    //=================================================================
    // 16 - Stack buffer conveyors
    //=================================================================

    // EN: Common speed reference for all stack buffer conveyors [m/min].
    // PT: Referência comum de velocidade para todas as esteiras buffer [m/min].
    stackBufferConveyorsSpeedMPM               : REAL := 20.0;

    // EN: Additional running time after the target sensor is activated
    //     on buffer conveyors 1 and 2. Conveyor 3 stops immediately.
    // PT: Tempo adicional de movimento após o acionamento do sensor alvo
    //     nas esteiras buffer 1 e 2. A esteira 3 para imediatamente.
    stackBufferConveyorsStopDelay              : TIME := T#500MS;

    // EN: Maximum time allowed to transfer a stack to a buffer position.
    // PT: Tempo máximo permitido para transferir uma pilha até uma posição buffer.
    stackBufferTransferTimeout                 : TIME := T#30S;

    // EN: Time with all buffer positions occupied before requesting
    //     a machine speed reduction.
    // PT: Tempo com todas as posições buffer ocupadas antes de solicitar
    //     a redução da velocidade da máquina.
    stackBufferFullSpeedReductionDelay         : TIME := T#10S;

	//==============================================================
	// Configuration parameters / Parâmetros de configuração
	//==============================================================
	paperPressOnTime  : TIME := T#2S;
	paperPressOffTime : TIME := T#6S;

    //=================================================================
    // 17 - EN: Elevator servo controlled shutdown
    //      PT: Desligamento controlado do servo do elevador
    //=================================================================

    // EN: Time to keep the elevator servo enabled while quick stop is processed.
    // PT: Tempo para manter o servo do elevador habilitado durante o processamento do quick stop.
    elevatorDriveDisableDelay          : TIME := T#500MS;

    //=================================================================
    // 18 - Sheet conveyor 1 exhaust fan
    //=================================================================

    // EN: Minimum line speed required to run the exhaust fan [m/min].
    // PT: Velocidade mínima da linha necessária para ligar o exaustor [m/min].
    sheetConveyor1ExhaustFanLineSpeedThresholdMPM : REAL := 10.0;

    // EN: Time to keep the exhaust fan running after line speed drops
    //     to or below the configured threshold.
    // PT: Tempo para manter o exaustor ligado após a velocidade da linha cair
    //     até ou abaixo do limite configurado.
    sheetConveyor1ExhaustFanStopDelay              : TIME := T#10S;

END_STRUCT
END_TYPE

// ---- Library/Machine/Stacker/Cpx/DataTypes/hmiAlarmsComplexStacker_TypeStruct.TcDUT
TYPE hmiAlarmsComplexStacker_TypeStruct :
STRUCT

    //==============================================================
    // General / system alarms
    //==============================================================
    safetyCircuitNotOk                 : BOOL;
    systemFaultActive                  : BOOL;
    systemNotEnabled                   : BOOL;

    // EN: Generic safety feedback diagnostic alarms.
    // PT: Alarmes genéricos de diagnóstico dos retornos de segurança.
    safetyFeedback1NotOk               : BOOL;
    safetyFeedback2NotOk               : BOOL;
    safetyFeedback3NotOk               : BOOL;
    safetyFeedback4NotOk               : BOOL;
    safetyFeedback5NotOk               : BOOL;
    safetyFeedback6NotOk               : BOOL;
    safetyFeedback7NotOk               : BOOL;
    safetyFeedback8NotOk               : BOOL;

    //==============================================================
    // Sheet conveyor group alarms
    //==============================================================
    sheetConveyor1DriveNotOk           : BOOL;
    sheetConveyor2DriveNotOk           : BOOL;
    sheetConveyor3DriveNotOk           : BOOL;
    sheetConveyor4DriveNotOk           : BOOL;
    sheetConveyorGroupFault            : BOOL;
    synchronizedConveyorsNotRunning    : BOOL;

    //==============================================================
    // EN: Stack buffer conveyor alarms
    // PT: Alarmes das esteiras buffer de pilhas
    //==============================================================
    stackBufferConveyor1DriveNotOk      : BOOL;
    stackBufferConveyor2DriveNotOk      : BOOL;
    stackBufferConveyor3DriveNotOk      : BOOL;
    stackBufferConveyorGroupFault       : BOOL;

    // EN: Automatic stack transfer exceeded the configured timeout.
    // PT: A transferência automática da pilha excedeu o timeout configurado.
    stackBufferTransferTimeout          : BOOL;

    // EN: All three stack buffer positions are occupied.
    // PT: As três posições do buffer de pilhas estão ocupadas.
    stackBufferFull                     : BOOL;

    // EN: Machine speed reduction was requested because the buffer stayed full.
    // PT: A redução de velocidade da máquina foi solicitada porque o buffer permaneceu cheio.
    stackBufferSpeedReductionActive     : BOOL;

    //==============================================================
    // Sheet stack separation alarms / indications
    //==============================================================
    sheetStackSeparationNotReady       : BOOL;
    sheetStackSeparationActive         : BOOL;
    sheetStackBrakeActive              : BOOL;

    //==============================================================
    // Sheet stack discharge sequence alarms / indications
    //==============================================================
    sheetStackDischargeFault           : BOOL;
    sheetStackDischargeLastCycleNotOk  : BOOL;
    sheetStackDischargeTimeout         : BOOL;
    sheetStackDischargeManualSkip      : BOOL;

    // EN: Detailed discharge sequence timeout alarms.
    // PT: Alarmes detalhados de timeout da sequência de descarte.
    sheetStackDischargeWaitSeparationTimeout : BOOL;
    sheetStackDischargePositioningTimeout    : BOOL;
    sheetStackDischargeConveyorStartTimeout  : BOOL;
    sheetStackDischargePlatformClearTimeout  : BOOL;
    sheetStackDischargeReturnTimeout         : BOOL;

    //==============================================================
    // Sheet stack discharge conveyor alarms
    //==============================================================
    sheetStackDischargeConveyorDriveNotOk : BOOL;
    sheetStackDischargeConveyorFault      : BOOL;

    //==============================================================
    // Backstop alarms / indications
    //==============================================================
    backstopDriveNotOk                 : BOOL;
    backstopFault                      : BOOL;
    backstopNotHomed                   : BOOL;
    backstopNotInPosition              : BOOL;

    // EN: Detailed backstop homing alarms.
    // PT: Alarmes detalhados do homing do backstop.
    backstopHomingTimeout              : BOOL;
    backstopInvalidHomeDirection       : BOOL;

    backstopSafeMaxLimitActive         : BOOL;
    backstopSafeMinLimitActive         : BOOL;
    backstopMaxLimitActive             : BOOL;
    backstopMinLimitActive             : BOOL;

    backstopManualInterventionActive   : BOOL;

    //==============================================================
    // Elevator alarms / indications
    //==============================================================
    elevatorDriveNotOk          : BOOL;
    elevatorFault               : BOOL;
    elevatorNotHomed            : BOOL;
    elevatorNotInPosition       : BOOL;

    // EN: Elevator homing exceeded the configured timeout.
    // PT: O homing do elevador excedeu o timeout configurado.
    elevatorHomingTimeout       : BOOL;

    // EN: An upward movement request is blocked by the backstop material sensor.
    // PT: Um pedido de subida está bloqueado pelo sensor de material do backstop.
    elevatorUpBlockedByBackstopMaterialInterlock : BOOL;

    elevatorUpperSafetyLimitActive : BOOL;
    elevatorLowerSafetyLimitActive : BOOL;
    elevatorUpperLimitActive       : BOOL;
    elevatorLowerLimitActive       : BOOL;

END_STRUCT
END_TYPE

// ---- Library/Machine/Stacker/Cpx/DataTypes/hmiCommandsComplexStacker_TypeStruct.TcDUT
TYPE hmiCommandsComplexStacker_TypeStruct :
STRUCT

    //==============================================================
    // EN: System master commands
    // PT: Comandos gerais do sistema
    //==============================================================
    // EN: Momentary master start command.
    // PT: Comando momentâneo de partida geral.
    startCmd                                : BOOL;

    // EN: Momentary master stop command.
    // PT: Comando momentâneo de parada geral.
    stopCmd                                 : BOOL;

    // EN: Momentary fault reset command.
    // PT: Comando momentâneo de reset das falhas.
    resetCmd                                : BOOL;

	blockConveyorCmd					: BOOL;

    //==============================================================
    // EN: Sheet conveyor group commands
    // PT: Comandos do grupo de esteiras de chapas
    //==============================================================
    // EN: Momentary speed-up command for the sheet conveyors.
    // PT: Comando momentâneo para acelerar as esteiras de chapas.
    sheetConveyorsSpeedUpCmd                : BOOL;


    //==============================================================
    // EN: Package and sheet handling commands
    // PT: Comandos de pacote e manuseio das chapas
    //==============================================================
    // EN: Momentary request to complete and discharge the current package.
    // PT: Solicitação momentânea para concluir e descarregar o pacote atual.
    packageCompleteCmd                      : BOOL;

    // EN: Command to lower the no-crush rollers.
    // PT: Comando para baixar os rolos no-crush.
    noCrushRollersDownCmd                   : BOOL;


    //==============================================================
    // EN: Elevator commands
    // PT: Comandos do elevador
    //==============================================================
    // EN: Maintained elevator automatic-mode command.
    // PT: Comando mantido do modo automático do elevador.
    elevatorAutoCmd                         : BOOL;

    // EN: Momentary elevator homing command.
    // PT: Comando momentâneo de homing do elevador.
    elevatorHomeCmd                         : BOOL;

    // EN: Hold-to-run elevator jog-up command.
    // PT: Comando de jog mantido para subir o elevador.
    elevatorUpCmd                           : BOOL;

    // EN: Hold-to-run elevator jog-down command.
    // PT: Comando de jog mantido para descer o elevador.
    elevatorDownCmd                         : BOOL;


    //==============================================================
    // EN: Backstop commands
    // PT: Comandos do backstop
    //==============================================================
    // EN: Maintained backstop automatic-mode command.
    // PT: Comando mantido do modo automático do backstop.
    backstopAutoCmd                         : BOOL;

    // EN: Momentary backstop homing command.
    // PT: Comando momentâneo de homing do backstop.
    backstopHomeCmd                         : BOOL;

    // EN: Momentary command to execute programmed backstop positioning.
    // PT: Comando momentâneo para executar o posicionamento programado do backstop.
    backstopExecutePositioningCmd           : BOOL;

    // EN: Hold-to-run command to open the backstop.
    // PT: Comando mantido de jog para abrir o backstop.
    backstopOpenCmd                         : BOOL;

    // EN: Hold-to-run command to close the backstop.
    // PT: Comando mantido de jog para fechar o backstop.
    backstopCloseCmd                        : BOOL;


    //==============================================================
    // EN: Discharge and stack buffer conveyor commands
    // PT: Comandos das esteiras de descarga e buffer de pilhas
    //==============================================================
    // EN: Hold-to-run manual command for the stack discharge conveyor.
    // PT: Comando manual mantido da esteira de descarga da pilha.
    sheetStackDischargeConveyorManualRunCmd : BOOL;

    // EN: Hold-to-run manual command for all stack buffer conveyors.
    // PT: Comando manual mantido para todas as esteiras buffer de pilhas.
    stackBufferConveyorsRunCmd              : BOOL;


    //==============================================================
    // EN: Auxiliary pneumatic commands
    // PT: Comandos pneumáticos auxiliares
    //==============================================================
    // EN: Enables the cyclic paper press operation.
    // PT: Habilita a operação cíclica do prensa-papel.
    paperPressAutoManCmd                    : BOOL;

    // EN: Enables automatic operation of the exhaust fan installed
    //     on sheet conveyor 1.
    // PT: Habilita a operação automática do exaustor instalado
    //     na esteira de chapas 1.
    sheetConveyor1ExhaustFanCmd             : BOOL;

    // EN: Enables the four independent sheet brush commands.
    // PT: Habilita os comandos independentes das quatro escovas de chapas.
    sheetBrushAutoManCmd                    : BOOL;

    // EN: Individual sheet brush commands.
    // PT: Comandos individuais das escovas de chapas.
    sheetBrush1Cmd                          : BOOL;
    sheetBrush2Cmd                          : BOOL;
    sheetBrush3Cmd                          : BOOL;
    sheetBrush4Cmd                          : BOOL;

END_STRUCT
END_TYPE

// ---- Library/Machine/Stacker/Cpx/DataTypes/hmiStatusComplexStacker_TypeStruct.TcDUT
TYPE hmiStatusComplexStacker_TypeStruct :
STRUCT

    //==============================================================
    // System general status
    //==============================================================
    systemRunEnable                         : BOOL;        // EN: Master system run enable
    safetyCircuitOk                         : BOOL;        // EN: Safety circuit status
    faultActive                             : BOOL;        // EN: General fault active
    deviceState                             : STRING(30);  // EN: General device state text


    //==============================================================
    // Sheet conveyor group status
    //==============================================================
    synchronizedConveyorsRunning            : BOOL;        // EN: All synchronized conveyors running

    sheetConveyor1Run                       : BOOL;        // EN: Sheet conveyor 1 run output
    sheetConveyor2Run                       : BOOL;        // EN: Sheet conveyor 2 run output
    sheetConveyor3Run                       : BOOL;        // EN: Sheet conveyor 3 run output
    sheetConveyor4Run                       : BOOL;        // EN: Sheet conveyor 4 run output

    sheetConveyor1SpeedRefMPM               : REAL;        // EN: Sheet conveyor 1 speed reference [m/min]
    sheetConveyor2SpeedRefMPM               : REAL;        // EN: Sheet conveyor 2 speed reference [m/min]
    sheetConveyor3SpeedRefMPM               : REAL;        // EN: Sheet conveyor 3 speed reference [m/min]
    sheetConveyor4SpeedRefMPM               : REAL;        // EN: Sheet conveyor 4 speed reference [m/min]

    syncConveyorsState                      : INT;         // EN: Synchronized conveyor group state code


    //==============================================================
    // Sheet stack separation status
    //==============================================================
    sheetStackSeparationReady               : BOOL;        // EN: Stack separation ready
    sheetStackSeparationActive              : BOOL;        // EN: Stack separation active
    sheetStackBrakeActive                   : BOOL;        // EN: Stack brake active

    sheetStackSeparationDistanceM           : REAL;        // EN: Current separation distance [m]
    sheetStackSeparationTargetDistanceM     : REAL;        // EN: Target separation distance [m]


    //==============================================================
    // Sheet stack discharge sequence status
    //==============================================================
    sheetStackDischargeState                : STRING(30);  // EN: Discharge sequence state text
    sheetStackDischargeStateCode            : INT;         // EN: Discharge sequence state code

    sheetStackDischargePending              : BOOL;        // EN: Discharge cycle pending
    sheetStackDischargeActive               : BOOL;        // EN: Discharge cycle active
    sheetStackDischargeStarted              : BOOL;        // EN: Discharge cycle started pulse/status
    sheetStackDischargeFinished             : BOOL;        // EN: Discharge cycle finished pulse/status

    sheetStackDischargeFault                : BOOL;        // EN: Discharge sequence fault
    sheetStackDischargeFaultCode            : INT;         // EN: Current discharge fault code

    sheetStackDischargeLastCycleOk          : BOOL;        // EN: Last discharge cycle completed successfully
    sheetStackDischargeLastResultCode       : INT;         // EN: Last discharge result code
    sheetStackDischargeLastFaultStepCode    : INT;         // EN: Last discharge fault step code
    sheetStackDischargeLastFaultCode        : INT;         // EN: Last discharge fault code


    //==============================================================
    // Sheet stack discharge conveyor status
    //==============================================================
    sheetStackDischargeConveyorState        : STRING(30);  // EN: Discharge conveyor state text
    sheetStackDischargeConveyorRun          : BOOL;        // EN: Discharge conveyor run output
    sheetStackDischargeConveyorSpeedRefMPM  : REAL;        // EN: Discharge conveyor speed reference [m/min]

    sheetStackDischargeConveyorFault        : BOOL;        // EN: Discharge conveyor fault
    sheetStackDischargeConveyorFaultCode    : INT;         // EN: Discharge conveyor fault code


    //==============================================================
    // Backstop status
    //==============================================================
    backstopState                           : STRING(30);  // EN: Backstop state text
    backstopHomed                           : BOOL;        // EN: Backstop homing completed
    backstopHomeRunning                     : BOOL;        // EN: Backstop homing sequence running
    backstopInPosition                      : BOOL;        // EN: Backstop is inside target tolerance

    backstopPositionMm                      : REAL;        // EN: Actual backstop position [mm]
    backstopTargetPositionMm                : REAL;        // EN: Active backstop target position [mm]
    backstopPositionErrorMm                 : REAL;        // EN: Backstop position error [mm]

    backstopRunFw                           : BOOL;        // EN: Backstop forward/open run output
    backstopRunRev                          : BOOL;        // EN: Backstop reverse/close run output
    backstopSpeedRefMmps                    : REAL;        // EN: Backstop speed reference [mm/s]

    backstopPlateUpSolenoid                 : BOOL;        // EN: Backstop plate up solenoid
    backstopSetEncoderPosition              : BOOL;        // EN: Backstop set encoder pulse
    backstopSetEncoderPositionMm            : REAL;        // EN: Backstop set encoder position [mm]

    backstopManualInterventionActive        : BOOL;        // EN: Manual intervention memory active
    backstopManualInterventionPositionMm    : REAL;        // EN: Stored manual intervention position [mm]

    backstopFault                           : BOOL;        // EN: Backstop fault
    backstopFaultCode                       : INT;         // EN: Backstop fault code


    //==============================================================
    // Elevator status
    //==============================================================
    elevatorState                    : STRING(30);  // EN: Elevator state text
    elevatorHomed                    : BOOL;        // EN: Elevator homing completed
    elevatorInPosition               : BOOL;        // EN: Elevator is inside target tolerance

    elevatorPositionMm               : REAL;        // EN: Actual elevator position [mm]
    elevatorTargetPositionMm         : REAL;        // EN: Active elevator target position [mm]
    elevatorPositionErrorMm          : REAL;        // EN: Elevator position error [mm]

    elevatorRunUp                    : BOOL;        // EN: Elevator up run output
    elevatorRunDown                  : BOOL;        // EN: Elevator down run output
    elevatorBrakeRelease             : BOOL;        // EN: Elevator brake release output

    // EN: Elevator servo enable and quick-stop outputs.
    // PT: Saídas de habilitação e quick stop do servo do elevador.
    elevatorDriveEnable               : BOOL;
    elevatorQuickStop                 : BOOL;

    elevatorSpeedRefMmps             : REAL;        // EN: Elevator speed reference [mm/s]

    elevatorSetEncoderPosition       : BOOL;        // EN: Elevator set encoder pulse
    elevatorSetEncoderPositionMm     : REAL;        // EN: Elevator set encoder position [mm]

    elevatorFault                    : BOOL;        // EN: Elevator fault
    elevatorFaultCode                : INT;         // EN: Elevator fault code


    //==============================================================
    // EN: Auxiliary pneumatic output status
    // PT: Estados das saídas pneumáticas auxiliares
    //==============================================================
    // EN: Paper press solenoid output.
    // PT: Saída do solenoide do prensa-papel.
    paperPressSolenoid                      : BOOL;

    // EN: Sheet conveyor 1 exhaust fan run output.
    // PT: Saída de acionamento do exaustor da esteira de chapas 1.
    sheetConveyor1ExhaustFanRun             : BOOL;

    // EN: Sheet brush valve outputs.
    // PT: Saídas das válvulas das escovas de chapas.
    sheetBrush1Valve                        : BOOL;
    sheetBrush2Valve                        : BOOL;
    sheetBrush3Valve                        : BOOL;
    sheetBrush4Valve                        : BOOL;


    //==============================================================
    // Process values
    //==============================================================
    lineSpeedMPM                            : REAL;        // EN: Current line speed [m/min]
    sheetLengthMm                           : REAL;        // EN: Current sheet length [mm]
    stackHeightMm                           : REAL;        // EN: Current stack height [mm]


    //==============================================================
    // Input / drive status mirror
    //==============================================================
    sheetConveyor1DriveOk                   : BOOL;        // EN: Sheet conveyor 1 drive OK
    sheetConveyor2DriveOk                   : BOOL;        // EN: Sheet conveyor 2 drive OK
    sheetConveyor3DriveOk                   : BOOL;        // EN: Sheet conveyor 3 drive OK
    sheetConveyor4DriveOk                   : BOOL;        // EN: Sheet conveyor 4 drive OK

    backstopDriveOk                         : BOOL;        // EN: Backstop drive OK
    elevatorDriveOk                  : BOOL;        // EN: Elevator drive OK
    sheetStackDischargeConveyorDriveOk      : BOOL;        // EN: Discharge conveyor drive OK

END_STRUCT
END_TYPE

// ---- Library/Machine/Stacker/Simple/DataTypes/SimpleStackerConfig_TypeStruct.TcDUT
TYPE SimpleStackerConfig_TypeStruct :
STRUCT

    //=================================================================
    // 01 - General line / stacker speed configuration
    //=================================================================

    // EN: Normal stacker speed ratio relative to line speed.
    //     Example: 0.17 = stacker runs at 17% of line speed.
    // PT: Fator normal de velocidade do stacker em relação à velocidade da linha.
    //     Exemplo: 0.17 = stacker trabalha com 17% da velocidade da linha.
    stackerSpeedRatio                         : REAL := 0.17;

    // EN: Minimum and maximum speed reference allowed for sheet conveyors [m/min].
    // PT: Referência mínima e máxima permitida para as esteiras de chapas [m/min].
    minimumSpeedMPM                           : REAL := 10.0;
    maximumSpeedMPM                           : REAL := 80.0;

    // EN: Maximum ramp velocity for conveyor speed references [m/min/s].
    // PT: Velocidade máxima da rampa para referências das esteiras [m/min/s].
    rampVelocityUpMaxMPMps                    : REAL := 1000.0;
    rampVelocityDownMaxMPMps                  : REAL := 1000.0;

    // EN: Ramp acceleration / deceleration used by S-ramp smoothing [m/min/s²].
    // PT: Aceleração / desaceleração usada na suavização da rampa S [m/min/s²].
    rampAccelerationUpMPMps2                  : REAL := 1000.0;
    rampAccelerationDownMPMps2                : REAL := 1000.0;


    //=================================================================
    // 02 - Sheet conveyor group: speed trim and mechanical length
    //=================================================================

    // EN: Individual speed trim for each synchronized sheet conveyor.
    //     1.0 = no correction.
    // PT: Correção individual de velocidade para cada esteira sincronizada.
    //     1.0 = sem correção.
    sheetConveyor1SpeedTrim                   : REAL := 1.0;
    sheetConveyor2SpeedTrim                   : REAL := 1.0;
    sheetConveyor3SpeedTrim                   : REAL := 1.0;

    // EN: Sheet conveyor mechanical length [m].
    // PT: Comprimento mecânico da esteira de chapas [m].
    sheetConveyor1LengthM                     : REAL := 1.85;
    sheetConveyor2LengthM                     : REAL := 1.0;
    sheetConveyor3LengthM                     : REAL := 2.0;

    // EN: Additional speed reference applied to sheet conveyors 1, 2 and 3
    //     when the external speed-up command is active [m/min].
    // PT: Referência adicional aplicada nas esteiras 1, 2 e 3
    //     quando o comando externo de aceleração estiver ativo [m/min].
    sheetConveyorsSpeedUpMPM                  : REAL := 20.0;


    //=================================================================
    // 03 - Sheet conveyor group: package separation
    //=================================================================

    // EN: Speed multiplier used during package separation.
    //     Example: 1.50 = 50% faster than normal speed.
    // PT: Multiplicador de velocidade usado durante a separação de pacote.
    //     Exemplo: 1.50 = 50% acima da velocidade normal.
    packageGapSpeedRatio                      : REAL := 3.0;

    // EN: Additional fixed speed offset during package separation [m/min].
    // PT: Offset fixo adicional de velocidade durante a separação de pacote [m/min].
    packageGapSpeedOffsetMPM                  : REAL := 0.0;

    // EN: Minimum line speed used as the conveyor speed calculation reference
    //     while package separation is active [m/min].
    //     Set to 0.0 to keep the actual line speed without a discharge override.
    // PT: Velocidade mínima da linha usada como referência para o cálculo das
    //     esteiras enquanto a separação da pilha estiver ativa [m/min].
    //     Usar 0.0 para manter a velocidade real da linha sem sobreposição no descarte.
    packageDischargeLineSpeedThresholdMPM     : REAL := 0.0;

    // EN: Minimum valid differential speed used for separation tracking [m/min].
    // PT: Velocidade diferencial mínima válida usada no rastreamento da separação [m/min].
    minimumOpeningSpeedMPM                    : REAL := 1.0;


    //=================================================================
    // 04 - Conveyor leveler: speed trim and position limits
    //=================================================================

    // EN: Individual speed trim for conveyor leveler synchronized movement.
    //     1.0 = no correction.
    // PT: Correção individual de velocidade para movimento sincronizado do nivelador.
    //     1.0 = sem correção.
    conveyorLevelerSpeedTrim                  : REAL := 1.0;

    // EN: Minimum and maximum allowed conveyor leveler position [mm].
    // PT: Posição mínima e máxima permitida para o nivelador da esteira [mm].
    conveyorLevelerMinPositionMm              : REAL := 10.0;
    conveyorLevelerMaxPositionMm              : REAL := 150.0;


    //=================================================================
    // 05 - Conveyor leveler: automatic positioning
    //=================================================================

    // EN: Offset added to stack height to calculate conveyor leveler target [mm].
    // PT: Offset somado à altura da pilha para calcular o alvo do nivelador [mm].
    conveyorLevelerStackHeightOffsetMm        : REAL := 0.0;

    // EN: Position tolerance to consider conveyor leveler in position [mm].
    // PT: Tolerância de posição para considerar o nivelador em posição [mm].
    conveyorLevelerPositionToleranceMm        : REAL := 2.0;

    // EN: Proportional gain for conveyor leveler position control [(mm/s)/mm].
    // PT: Ganho proporcional do controle de posição do nivelador [(mm/s)/mm].
    conveyorLevelerPositionKp                 : REAL := 5.0;

    // EN: Maximum speed allowed in automatic conveyor leveler positioning [mm/s].
    // PT: Velocidade máxima permitida no posicionamento automático do nivelador [mm/s].
    conveyorLevelerAutoMaxSpeedMmps           : REAL := 30.0;

    // EN: Minimum movement speed when the position error is above tolerance [mm/s].
    // PT: Velocidade mínima de movimento quando o erro de posição estiver acima da tolerância [mm/s].
    conveyorLevelerMinMoveSpeedMmps           : REAL := 5.0;


    //=================================================================
    // 06 - Conveyor leveler: manual movement
    //=================================================================

    // EN: Manual up/down speed for conveyor leveler [mm/s].
    // PT: Velocidade manual para subir/descer o nivelador da esteira [mm/s].
    conveyorLevelerManualSpeedMmps            : REAL := 50.0;

    // EN: Minimum speed reference required to enable conveyor leveler drive run [mm/s].
    // PT: Referência mínima de velocidade necessária para liberar RUN do acionamento do nivelador [mm/s].
    conveyorLevelerRunMinSpeedMmps            : REAL := 0.1;


    //=================================================================
    // 07 - Conveyor leveler: homing and encoder set
    //=================================================================

    // EN: Conveyor leveler homing speed [mm/s].
    // PT: Velocidade de homing do nivelador da esteira [mm/s].
    conveyorLevelerHomingSpeedMmps            : REAL := 30.0;

    // EN: Maximum allowed time for conveyor leveler homing movement.
    // PT: Tempo máximo permitido para o movimento de homing do nivelador.
    conveyorLevelerHomingTimeout              : TIME := T#30S;

    // EN: Pulse time for conveyor leveler encoder position set command.
    // PT: Tempo do pulso para comando de set da posição do encoder do nivelador.
    conveyorLevelerSetEncoderPulseTime        : TIME := T#200MS;


    //=================================================================
    // 08 - Conveyor leveler: magnetic brake
    //=================================================================

    // EN: Delay between brake release command and motor movement permission.
    // PT: Atraso entre o comando de liberação do freio e a permissão de movimento do motor.
    conveyorLevelerBrakeReleaseDelay          : TIME := T#300MS;

    // EN: Time to keep the brake released after movement stops.
    // PT: Tempo para manter o freio liberado após a parada do movimento.
    conveyorLevelerBrakeHoldTime              : TIME := T#2S;


    //=================================================================
    // 09 - Backstop: position limits
    //=================================================================

    // EN: Minimum and maximum allowed backstop position [mm].
    // PT: Posição mínima e máxima permitida para o backstop [mm].
    backstopMinPositionMm                     : REAL := 300.0;
    backstopMaxPositionMm                     : REAL := 5000.0;


    //=================================================================
    // 10 - Backstop: homing and encoder set
    //=================================================================

    // EN: Homing direction. -1 = close/min limit, +1 = open/max limit.
    // PT: Direção de homing. -1 = fechar/limite mínimo, +1 = abrir/limite máximo.
    backstopHomeDirection                     : INT := 1;

    // EN: Encoder position value to set after homing is completed [mm].
    // PT: Valor de posição gravado no encoder após finalizar o homing [mm].
    backstopHomePositionMm                    : REAL := 2985.0;

    // EN: Backstop homing speed [mm/s].
    // PT: Velocidade de homing do backstop [mm/s].
    backstopHomingSpeedMmps                   : REAL := 150.0;

    // EN: Maximum allowed time for backstop homing movement.
    // PT: Tempo máximo permitido para o movimento de homing do backstop.
    backstopHomingTimeout                     : TIME := T#40S;

    // EN: Pulse time for backstop encoder position set command.
    // PT: Tempo do pulso para comando de set da posição do encoder do backstop.
    backstopSetEncoderPulseTime               : TIME := T#200MS;


    //=================================================================
    // 11 - Backstop: automatic positioning
    //=================================================================

    // EN: Offset added to sheet length to calculate automatic backstop target [mm].
    // PT: Offset somado ao comprimento da chapa para calcular o alvo automático do backstop [mm].
    backstopSheetLengthOffsetMm               : REAL := 0.0;

    // EN: Position tolerance to consider the backstop in position [mm].
    // PT: Tolerância de posição para considerar o backstop em posição [mm].
    backstopPositionToleranceMm               : REAL := 5.0;

    // EN: Proportional gain for backstop position control [(mm/s)/mm].
    // PT: Ganho proporcional do controle de posição do backstop [(mm/s)/mm].
    backstopPositionKp                        : REAL := 3.0;

    // EN: Maximum speed allowed in automatic backstop positioning [mm/s].
    // PT: Velocidade máxima permitida no posicionamento automático do backstop [mm/s].
    backstopAutoMaxSpeedMmps                  : REAL := 400.0;

    // EN: Minimum movement speed when the position error is above tolerance [mm/s].
    // PT: Velocidade mínima de movimento quando o erro de posição estiver acima da tolerância [mm/s].
    backstopMinMoveSpeedMmps                  : REAL := 15.0;


    //=================================================================
    // 12 - Backstop: manual movement
    //=================================================================

    // EN: Manual open/close speed for backstop [mm/s].
    // PT: Velocidade manual para abrir/fechar o backstop [mm/s].
    backstopManualSpeedMmps                   : REAL := 80.0;

    // EN: Minimum speed reference required to enable backstop drive run [mm/s].
    // PT: Referência mínima de velocidade necessária para liberar RUN do acionamento do backstop [mm/s].
    backstopRunMinSpeedMmps                   : REAL := 10.0;


    //=================================================================
    // 13 - Sheet stack discharge conveyor
    //=================================================================

    // EN: Sheet stack discharge conveyor speed reference [m/min].
    // PT: Referência de velocidade da esteira de descarga da pilha [m/min].
    sheetStackDischargeConveyorSpeedMPM       : REAL := 70.0;

    // EN: Running time for sheet stack discharge conveyor.
    // PT: Tempo de giro da esteira de descarga da pilha.
    sheetStackDischargeTime                   : TIME := T#2S;


    //=================================================================
    // 14 - Sheet stack discharge sequence: backstop movement
    //=================================================================

    // EN: Additional backstop opening during sheet stack discharge [mm].
    // PT: Abertura adicional do backstop durante a descarga da pilha [mm].
    backstopDischargeOpenOffsetMm             : REAL := 100.0;


    //=================================================================
    // 15 - Sheet stack discharge sequence: step timeouts
    //=================================================================

    // EN: Maximum time to wait for package separation before discharge sequence continues.
    // PT: Tempo máximo de espera pela separação do pacote antes da sequência de descarga continuar.
    sheetStackDischargeWaitSeparationTimeout  : TIME := T#10S;

    // EN: Maximum time allowed for discharge positioning movement.
    // PT: Tempo máximo permitido para o movimento de posicionamento da descarga.
    sheetStackDischargePositioningTimeout     : TIME := T#10S;

    // EN: Maximum time allowed to confirm/start discharge conveyor movement.
    // PT: Tempo máximo permitido para confirmar/iniciar o movimento da esteira de descarga.
    sheetStackDischargeConveyorStartTimeout   : TIME := T#3S;

    // EN: Maximum time allowed for backstop return movement after discharge.
    // PT: Tempo máximo permitido para o retorno do backstop após a descarga.
    sheetStackDischargeReturnTimeout          : TIME := T#10S;

END_STRUCT
END_TYPE

// ---- Library/Machine/Stacker/Simple/DataTypes/SimpleStackerConfig_TypeStruct_1.TcDUT
TYPE SimpleStackerConfig_TypeStruct_1 :
STRUCT

    //==============================================================
    // Normal speed synchronization
    //==============================================================
    // EN: Normal stacker speed ratio relative to line speed.
    //     Example: 0.17 = stacker runs at 17% of line speed.
    // PT: Fator normal de velocidade do stacker em relação à linha.
    //     Exemplo: 0.17 = stacker trabalha com 17% da velocidade da linha.
    stackerSpeedRatio                 : REAL := 0.17;


    //==============================================================
    // Individual conveyor speed trim
    //==============================================================
    // EN: Individual speed correction for each conveyor.
    // PT: Correção individual de velocidade de cada esteira.
    sheetConveyor1SpeedTrim           : REAL := 1.0;
    sheetConveyor2SpeedTrim           : REAL := 1.0;
    sheetConveyor3SpeedTrim           : REAL := 1.0;
    conveyorLevelerSpeedTrim          : REAL := 1.0;

	//==============================================================
	// Sheet conveyors speed-up command
	//==============================================================
	// EN: Additional speed reference applied to sheet conveyors 1/2/3 [m/min].
	// PT: Referência adicional aplicada nas esteiras 1/2/3 [m/min].
	sheetConveyorsSpeedUpMPM : REAL := 20.0;
	
    //==============================================================
    // Conveyor length
    //==============================================================
    // EN: Conveyor length [m].
    // PT: Comprimento da esteira [m].
    sheetConveyor1LengthM             : REAL := 20.0;
    sheetConveyor2LengthM             : REAL := 20.0;
    sheetConveyor3LengthM             : REAL := 20.0;


    //==============================================================
    // Package separation
    //==============================================================
    // EN: Speed multiplier used during package separation.
    // PT: Multiplicador de velocidade usado durante a separação.
    packageGapSpeedRatio              : REAL := 1.50;

    // EN: Additional fixed speed offset during separation [m/min].
    // PT: Offset fixo adicional de velocidade durante a separação [m/min].
    packageGapSpeedOffsetMPM          : REAL := 0.0;

    // EN: Gap distance as factor of sheet length.
    //     Example: 0.25 with 2.0 m sheet = 0.5 m gap.
    // PT: Distância de abertura como fator do comprimento da chapa.
    //     Exemplo: 0.25 com chapa de 2.0 m = 0.5 m de vão.
//    packageGapLengthFactor            : REAL := 0.25;

    // EN: Minimum valid differential speed for opening calculation [m/min].
    // PT: Velocidade diferencial mínima válida para cálculo de abertura [m/min].
    minimumOpeningSpeedMPM            : REAL := 1.0;

    // EN: Maximum package gap distance allowed [m].
    // PT: Distância máxima permitida para abertura do pacote [m].
//    maximumPackageGapDistanceM        : REAL := 3.0;


    //==============================================================
    // Speed limits
    //==============================================================
    // EN: Minimum and maximum conveyor speed reference [m/min].
    // PT: Velocidade mínima e máxima de referência das esteiras [m/min].
    minimumSpeedMPM                   : REAL := 0.0;
    maximumSpeedMPM                   : REAL := 80.0;


    //==============================================================
    // Ramp parameters
    //==============================================================
    // EN: Maximum ramp velocity [m/min/s].
    // PT: Velocidade máxima da rampa [m/min/s].
    rampVelocityUpMaxMPMps            : REAL := 1000.0;
    rampVelocityDownMaxMPMps          : REAL := 1000.0;

    // EN: Ramp acceleration / S-ramp smoothing [m/min/s²].
    // PT: Aceleração da rampa / suavização da rampa S [m/min/s²].
    rampAccelerationUpMPMps2          : REAL := 1000.0;
    rampAccelerationDownMPMps2        : REAL := 1000.0;



	//==============================================================
	// Backstop homing
	//==============================================================
	// EN: Homing direction. -1 = close/min limit, +1 = open/max limit.
	// PT: Direção de homing. -1 = fechar/limite mínimo, +1 = abrir/limite máximo.
	backstopHomeDirection              : INT := -1;
	
	// EN: Encoder position value to set after homing is completed [mm].
	// PT: Valor de posição que será gravado no encoder após finalizar o homing [mm].
	backstopHomePositionMm             : REAL := 300.0;
	
	// EN: Backstop homing speed [mm/s].
	// PT: Velocidade de homing do backstop [mm/s].
	backstopHomingSpeedMmps            : REAL := 50.0;
	
	// EN: Maximum allowed time for homing movement.
	// PT: Tempo máximo permitido para o movimento de homing.
	backstopHomingTimeout              : TIME := T#30S;
	
	// EN: Pulse time for encoder position set command.
	// PT: Tempo do pulso para comando de set da posição do encoder.
	backstopSetEncoderPulseTime        : TIME := T#200MS;	
	//==============================================================
	// Backstop position limits
	//==============================================================
	// EN: Minimum allowed backstop position [mm].
	// PT: Posição mínima permitida do backstop [mm].
	backstopMinPositionMm              : REAL := 300.0;
	
	// EN: Maximum allowed backstop position [mm].
	// PT: Posição máxima permitida do backstop [mm].
	backstopMaxPositionMm              : REAL := 2500.0;
	
	
	//==============================================================
	// Backstop automatic positioning
	//==============================================================
	// EN: Offset added to sheet length to calculate automatic backstop target [mm].
	// PT: Offset somado ao comprimento da chapa para calcular o alvo automático [mm].
	backstopSheetLengthOffsetMm        : REAL := 0.0;
	
	// EN: Position tolerance to consider the backstop in position [mm].
	// PT: Tolerância de posição para considerar o backstop em posição [mm].
	backstopPositionToleranceMm        : REAL := 2.0;
	
	// EN: Proportional gain for position control [(mm/s)/mm].
	// PT: Ganho proporcional do controle de posição [(mm/s)/mm].
	backstopPositionKp                 : REAL := 0.5;
	
	// EN: Maximum speed allowed in automatic positioning [mm/s].
	// PT: Velocidade máxima permitida no posicionamento automático [mm/s].
	backstopAutoMaxSpeedMmps           : REAL := 150.0;
	
	// EN: Minimum movement speed when position error is above tolerance [mm/s].
	// PT: Velocidade mínima de movimento quando o erro de posição estiver acima da tolerância [mm/s].
	backstopMinMoveSpeedMmps           : REAL := 10.0;
	
	
	//==============================================================
	// Backstop manual movement
	//==============================================================
	// EN: Manual open/close speed [mm/s].
	// PT: Velocidade manual para abrir/fechar o backstop [mm/s].
	backstopManualSpeedMmps            : REAL := 80.0;
	
	// EN: Minimum speed reference to enable backstop drive run [mm/s].
	// PT: Referência mínima de velocidade para liberar RUN do inversor do backstop [mm/s].
	backstopRunMinSpeedMmps             : REAL := 0.1;
	
		
	//==============================================================
	// Conveyor leveler position limits
	//==============================================================
	conveyorLevelerMinPositionMm          : REAL := 0.0;
	conveyorLevelerMaxPositionMm          : REAL := 1000.0;
	
	
	//==============================================================
	// Conveyor leveler automatic control
	//==============================================================
	conveyorLevelerStackHeightOffsetMm    : REAL := 0.0;
	conveyorLevelerPositionToleranceMm    : REAL := 5.0;
	conveyorLevelerPositionKp             : REAL := 0.5;
	conveyorLevelerAutoMaxSpeedMmps       : REAL := 100.0;
	conveyorLevelerMinMoveSpeedMmps       : REAL := 5.0;
	
	
	//==============================================================
	// Conveyor leveler manual control
	//==============================================================
	conveyorLevelerManualSpeedMmps        : REAL := 50.0;
	
	
	//==============================================================
	// Conveyor leveler homing
	//==============================================================
	conveyorLevelerHomingSpeedMmps        : REAL := 30.0;
	conveyorLevelerHomingTimeout          : TIME := T#30S;
	
	
	//==============================================================
	// Conveyor leveler encoder set pulse
	//==============================================================
	conveyorLevelerSetEncoderPulseTime    : TIME := T#200MS;
	
	
	//==============================================================
	// Conveyor leveler magnetic brake
	//==============================================================
	conveyorLevelerBrakeReleaseDelay      : TIME := T#300MS;
	conveyorLevelerBrakeHoldTime          : TIME := T#2S;
	
	
	//==============================================================
	// Conveyor leveler drive enable
	//==============================================================
	conveyorLevelerRunMinSpeedMmps        : REAL := 0.1;	
	
	//==============================================================
	// Sheet stack discharge conveyor
	//==============================================================
	// EN: Discharge conveyor speed reference [m/min].
	// PT: Referência de velocidade da esteira de descarga [m/min].
	sheetStackDischargeConveyorSpeedMPM     : REAL := 20.0;
	
	// EN: Discharge conveyor running time.
	// PT: Tempo de giro da esteira de descarga.
	sheetStackDischargeTime                 : TIME := T#5S;
	
	
	//==============================================================
	// Backstop discharge movement
	//==============================================================
	// EN: Additional backstop opening during sheet stack discharge [mm].
	// PT: Abertura adicional do backstop durante a descarga da pilha [mm].
	backstopDischargeOpenOffsetMm           : REAL := 100.0;
	
	sheetStackDischargeWaitSeparationTimeout : TIME := T#10S;
	sheetStackDischargePositioningTimeout    : TIME := T#10S;
	sheetStackDischargeConveyorStartTimeout  : TIME := T#3S;
	sheetStackDischargeReturnTimeout         : TIME := T#10S;	
	
END_STRUCT
END_TYPE

// ---- Library/Machine/Stacker/Simple/E_BackstopState.TcDUT
{attribute 'qualified_only' := ''}
{attribute 'strict' := ''}
TYPE E_BackstopState :
(
	STOP := 0,
	HOME_FAST_SEARCH := 10,
	HOME_SLOW_EXIT_SENSOR := 11,
	HOME_SET_ENCODER := 12,
	HOME_WAIT_AFTER_SET := 13,
	HOME_MOVE_TO_TARGET := 14,
	MANUAL := 20,
	AUTO_POSITION := 30,
	FAULT := 40
);
END_TYPE

// ---- Library/Machine/Stacker/Simple/E_ConveyorLevelerState.TcDUT
{attribute 'qualified_only' := ''}
{attribute 'strict' := ''}
TYPE E_ConveyorLevelerState :
(
	STOP := 0,
	HOME_FAST_SEARCH := 10,
	HOME_SLOW_EXIT_SENSOR := 11,
	HOME_SET_ENCODER := 12,
	MANUAL := 20,
	AUTO_LEVELING := 30,
	FAULT := 40
);
END_TYPE

// ---- Library/Machine/Stacker/Simple/E_PackageSeparationState.TcDUT
{attribute 'qualified_only' := ''}
{attribute 'strict' := ''}
TYPE E_PackageSeparationState :
(
	NORMAL := 0,
	START_SEPARATION := 10,
	CONVEYOR_2_TRACKING := 20,
	CONVEYOR_3_TRACKING := 30,
	FINISH_SEPARATION := 40
);
END_TYPE

// ---- Library/Machine/Stacker/Simple/E_SheetStackDischargeState.TcDUT
{attribute 'qualified_only' := ''}
{attribute 'strict' := ''}
TYPE E_SheetStackDischargeState :
(
	IDLE := 0,
	WAIT_SEPARATION := 5,
	START_POSITIONING := 10,
	WAIT_BACKSTOP_POSITION := 20,
	DISCHARGING := 30,
	START_RETURN := 40,
	WAIT_BACKSTOP_RETURN := 50,
	FINISH := 60
);
END_TYPE

// ---- Library/Machine/Stacker/Simple/E_SyncConveyorsState.TcDUT
{attribute 'qualified_only' := ''}
{attribute 'strict' := ''}
TYPE E_SyncConveyorsState :
(
	IDLE := 0,
	RUN := 1,
	FAULT := 10
);
END_TYPE

// ---- Library/Sick/DT35-B15251 - Laser Sensor/DataTypes/_DT35B15251_DEV_CONFIG.TcDUT
TYPE _DT35B15251_DEV_CONFIG :
STRUCT

    //=============================================================
    // IO-Link process data
    //=============================================================

    processDataResolutionFactor : REAL := 1.0; 
    // 1.0 = process data in 1 mm steps
    // 0.1 = process data in 0.1 mm steps
    // 10.0 = process data in 10 mm steps


    //=============================================================
    // Distance limits
    //=============================================================

    distanceLowLimit  : REAL := 0.0;
    distanceHighLimit : REAL := 12000.0;


    //=============================================================
    // Relative distance from zero
    // EN: Shows distance starting from a configured zero point.
    // Example:
    // distance = 1500 mm
    // distanceZeroReference = 1000 mm
    // distanceFromZero = 500 mm
    //=============================================================

    distanceZeroReference       : REAL := 0.0;
    distanceFromZeroLowLimit    : REAL := 0.0;
    distanceFromZeroHighLimit   : REAL := 12000.0;


    //=============================================================
    // Height calculation
    // EN: Height is calculated from the measured distance.
    // Example:
    // heightReferenceDistance = distance from sensor to zero-height surface
    // height = heightReferenceDistance - distance
    //=============================================================

    heightReferenceDistance : REAL := 2000.0;
    heightLowLimit          : REAL := 0.0;
    heightHighLimit         : REAL := 2000.0;

END_STRUCT
END_TYPE

// ---- Library/Sick/DT35-B15251 - Laser Sensor/DataTypes/_DT35B15251_HWTOPLC_PDOS.TcDUT
TYPE _DT35B15251_HWTOPLC_PDOS :
STRUCT
	
	inputByte_0 	 : BYTE;
	inputByte_1 	 : BYTE;

END_STRUCT
END_TYPE

// ---- Library/Inovance/IS620P-CO/DataTypes/E_IS620P_CO_STATE.TcDUT
TYPE E_IS620P_CO_STATE :
(
    // EN: Function block execution is disabled.
    // PT: A execução do function block está desabilitada.
    Disabled,

    // EN: CANopen node or PDO feedback is not available.
    // PT: O nó CANopen ou a realimentação dos PDOs não está disponível.
    CommunicationFault,

    // EN: CiA 402 state: drive is not ready to switch on.
    // PT: Estado CiA 402: drive não está pronto para habilitação.
    NotReadyToSwitchOn,

    // EN: CiA 402 state: switch-on is disabled.
    // PT: Estado CiA 402: habilitação está desativada.
    SwitchOnDisabled,

    // EN: CiA 402 state: drive is ready to switch on.
    // PT: Estado CiA 402: drive está pronto para habilitação.
    ReadyToSwitchOn,

    // EN: CiA 402 state: drive is switched on.
    // PT: Estado CiA 402: drive está habilitado sem operação ativa.
    SwitchedOn,

    // EN: CiA 402 state: operation is enabled.
    // PT: Estado CiA 402: operação está habilitada.
    OperationEnabled,

    // EN: CiA 402 state: quick stop is active.
    // PT: Estado CiA 402: quick stop está ativo.
    QuickStopActive,

    // EN: CiA 402 state: fault reaction is active.
    // PT: Estado CiA 402: reação à falha está ativa.
    FaultReactionActive,

    // EN: CiA 402 state: drive has an active fault.
    // PT: Estado CiA 402: drive possui uma falha ativa.
    Fault
);
END_TYPE

// ---- Library/Inovance/IS620P-CO/DataTypes/IS620P_CO_DEV_CONFIG.TcDUT
TYPE IS620P_CO_DEV_CONFIG :
STRUCT
    // EN: Number of raw position units that represent one millimeter.
    // PT: Quantidade de unidades brutas de posição que representam um milímetro.
    positionUnitsPerMm       : LREAL := 1.0;

    // EN: Number of raw velocity units that represent one millimeter per second.
    // PT: Quantidade de unidades brutas de velocidade que representam um milímetro por segundo.
    velocityUnitsPerMmps     : LREAL := 1.0;

    // EN: Persistent offset applied to the converted position feedback.
    // PT: Offset persistente aplicado à realimentação de posição convertida.
    positionOffsetMm         : LREAL := 0.0;

    // EN: Indicates that a valid position calibration has been captured.
    // PT: Indica que uma calibração válida de posição foi capturada.
    calibrationValid         : BOOL := FALSE;

    // EN: Absolute equipment velocity limit applied before raw conversion.
    // PT: Limite absoluto de velocidade do equipamento aplicado antes da conversão bruta.
    maximumVelocityMmps      : LREAL := 100.0;

    // EN: Raw acceleration limit written to object 6083h.
    // PT: Limite bruto de aceleração escrito no objeto 6083h.
    profileAccelerationRaw   : UDINT := 100;

    // EN: Raw deceleration limit written to object 6084h.
    // PT: Limite bruto de desaceleração escrito no objeto 6084h.
    profileDecelerationRaw   : UDINT := 100;

    // EN: Reverses command and feedback signs when the mechanical direction is inverted.
    // PT: Inverte os sinais de comando e realimentação quando o sentido mecânico está invertido.
    directionInverted        : BOOL := FALSE;

    // EN: Maximum feedback velocity allowed when capturing a position calibration.
    // PT: Velocidade máxima de realimentação permitida ao capturar uma calibração de posição.
    positionSetMaxVelocityMmps : LREAL := 0.5;

    // EN: Maximum time allowed for drive enable sequencing.
    // PT: Tempo máximo permitido para a sequência de habilitação do drive.
    enableTimeout            : TIME := T#5S;

    // EN: Maximum time allowed to confirm Profile Velocity mode.
    // PT: Tempo máximo permitido para confirmar o modo Profile Velocity.
    modeSelectionTimeout     : TIME := T#5S;
END_STRUCT
END_TYPE

// ---- Library/Inovance/IS620P-CO/DataTypes/IS620P_CO_HWTOPLC_PDOS.TcDUT
{attribute 'pack_mode' := '1'}
TYPE IS620P_CO_HWTOPLC_PDOS :
STRUCT
	
    // EN: CiA 402 status word received from object 6041h.
    // PT: Palavra de estado CiA 402 recebida do objeto 6041h.
    statusWord      : UINT;

    // EN: Active operation mode received from object 6061h.
    // PT: Modo de operação ativo recebido do objeto 6061h.
    modeDisplay     : SINT;

    // EN: Raw position feedback received from object 6064h.
    // PT: Realimentação bruta de posição recebida do objeto 6064h.
    actualPosition  : DINT;

    // EN: Raw velocity feedback received from object 606Ch.
    // PT: Realimentação bruta de velocidade recebida do objeto 606Ch.
    actualVelocity  : DINT;

    // EN: CANopen node state supplied by the TwinCAT CANopen master at byte 11.
    // PT: Estado do nó CANopen fornecido pelo mestre CANopen do TwinCAT no byte 11.
    nodeState : USINT;

    // EN: Reserved hardware input bytes between NodeState and DiagFlag.
    // PT: Bytes reservados de entrada de hardware entre NodeState e DiagFlag.
    {attribute 'hide'}
    _reservedDiagnosticBytes : ARRAY [0..4] OF BYTE;

    // EN: Reserved hardware input bit immediately before DiagFlag.
    // PT: Bit reservado de entrada de hardware imediatamente antes de DiagFlag.
    {attribute 'hide'}
    _reservedDiagnosticBit : BIT;

    // EN: CANopen diagnostic-change flag supplied by the TwinCAT master at bit 137.
    // PT: Indicador de alteração de diagnóstico CANopen fornecido pelo mestre TwinCAT no bit 137.
    diagFlag : BIT;

    // EN: Remaining reserved bits in the CANopen diagnostic byte.
    // PT: Bits reservados restantes no byte de diagnóstico CANopen.
    {attribute 'hide'}
    _reservedDiagnosticBits : ARRAY [2..7] OF BOOL;
	
END_STRUCT
END_TYPE

// ---- Library/Inovance/IS620P-CO/DataTypes/IS620P_CO_PLCTOHW_PDOS.TcDUT
{attribute 'pack_mode' := '1'}
TYPE IS620P_CO_PLCTOHW_PDOS :
STRUCT
    // EN: CiA 402 control word sent to object 6040h.
    // PT: Palavra de controle CiA 402 enviada ao objeto 6040h.
    controlWord          : UINT;

    // EN: Requested operation mode sent to object 6060h.
    // PT: Modo de operação solicitado enviado ao objeto 6060h.
    modeCommand          : SINT;

    // EN: Position target mapped at object 607Ah and reserved for other modes.
    // PT: Alvo de posição mapeado no objeto 607Ah e reservado para outros modos.
    targetPosition       : DINT;

    // EN: Profile velocity mapped at object 6081h and reserved for other modes.
    // PT: Velocidade de perfil mapeada no objeto 6081h e reservada para outros modos.
    profileVelocity      : UDINT;

    // EN: Drive acceleration limit sent to object 6083h.
    // PT: Limite de aceleração do drive enviado ao objeto 6083h.
    profileAcceleration  : UDINT;

    // EN: Drive deceleration limit sent to object 6084h.
    // PT: Limite de desaceleração do drive enviado ao objeto 6084h.
    profileDeceleration  : UDINT;

    // EN: Signed velocity reference sent to object 60FFh.
    // PT: Referência de velocidade com sinal enviada ao objeto 60FFh.
    targetVelocity       : DINT;
END_STRUCT
END_TYPE

// ---- Library/Inovance/IS620P-CO/DataTypes/IS620P_CO_STATUS.TcDUT
TYPE IS620P_CO_STATUS :
STRUCT
    // EN: CANopen node and cyclic feedback are available.
    // PT: O nó CANopen e a realimentação cíclica estão disponíveis.
    communicationOk        : BOOL;

    // EN: Drive is ready to accept a velocity reference.
    // PT: O drive está pronto para aceitar uma referência de velocidade.
    ready                  : BOOL;

    // EN: CiA 402 Operation Enabled state is active.
    // PT: O estado CiA 402 Operation Enabled está ativo.
    driveEnabled           : BOOL;

    // EN: CiA 402 quick-stop state is active.
    // PT: O estado de quick stop CiA 402 está ativo.
    quickStopActive        : BOOL;

    // EN: Position feedback has a valid application offset.
    // PT: A realimentação de posição possui um offset válido da aplicação.
    calibrated             : BOOL;

    // EN: Drive reports a warning condition.
    // PT: O drive informa uma condição de advertência.
    warning                : BOOL;

    // EN: Drive reports a fault condition.
    // PT: O drive informa uma condição de falha.
    fault                  : BOOL;

    // EN: Device scaling parameters are valid.
    // PT: Os parâmetros de escala do equipamento são válidos.
    configurationValid     : BOOL;

    // EN: Drive enable sequence exceeded its configured timeout.
    // PT: A sequência de habilitação do drive excedeu o timeout configurado.
    enableTimeout          : BOOL;

    // EN: Profile Velocity mode confirmation exceeded its configured timeout.
    // PT: A confirmação do modo Profile Velocity excedeu o timeout configurado.
    modeSelectionTimeout   : BOOL;

    // EN: Raw CANopen node state supplied by the TwinCAT master.
    // PT: Estado bruto do nó CANopen fornecido pelo mestre TwinCAT.
    nodeState              : USINT;

    // EN: Indicates that CANopen diagnostic data changed.
    // PT: Indica que os dados de diagnóstico CANopen foram alterados.
    diagnosticFlag         : BOOL;

    // EN: Raw CiA 402 status word for diagnostics.
    // PT: Palavra de estado CiA 402 bruta para diagnóstico.
    statusWord             : UINT;

    // EN: Active operation mode reported by the drive.
    // PT: Modo de operação ativo informado pelo drive.
    activeMode             : SINT;

    // EN: Decoded generic device state.
    // PT: Estado genérico decodificado do equipamento.
    deviceState            : E_IS620P_CO_STATE;
END_STRUCT
END_TYPE

// ---- GVLs/GVL_Hmi.TcGVL
{attribute 'Tc2GvlVarNames'}
VAR_GLOBAL

	hmiCommands			: hmiCommands_TypeStruct;
	hmiStatus			: hmiStatus_TypeStruct;
	hmiAlarms			: hmiAlarms_TypeStruct;	

	
	
END_VAR

VAR_GLOBAL PERSISTENT

	machineConfig						: machineConfig_TypeStruct;
	currentOrder						: Order_TypeStruct;
	nextOrder							: Order_TypeStruct;
	hmiOrderStatus						: orderHmiStatus_TypeStruct;
	hmiOrderConfig						: orderConfig_TypeStruct;

END_VAR

// ---- GVLs/GVL_Hw.TcGVL
{attribute 'Tc2GvlVarNames'}
VAR_GLOBAL

	SLT1_P1_100_UG1		: AXIS_REF; //Knife 1 - axis variables
	SLT1_P1_100_UG2		: AXIS_REF; //Knife 2 - axis variables
	SLT1_P1_100_UG3		: AXIS_REF; //Knife 3 - axis variables
	SLT1_P1_100_UG4		: AXIS_REF; //Knife 4 - axis variables
	SLT1_P1_100_UG5		: AXIS_REF; //Knife 5 - axis variables
	SLT1_P1_100_UG6		: AXIS_REF; //Knife 6 - axis variables

	SLT1_P1_200_UG1		: AXIS_REF; //Scorer 1 - axis variables
	SLT1_P1_200_UG2		: AXIS_REF; //Scorer 2 - axis variables
	SLT1_P1_200_UG3		: AXIS_REF; //Scorer 3 - axis variables
	SLT1_P1_200_UG4		: AXIS_REF; //Scorer 4 - axis variables
	SLT1_P1_200_UG5		: AXIS_REF; //Scorer 5 - axis variables
	SLT1_P1_200_UG6		: AXIS_REF; //Scorer 6 - axis variables
	SLT1_P1_200_UG7		: AXIS_REF; //Scorer 7 - axis variables
	SLT1_P1_200_UG8		: AXIS_REF; //Scorer 8 - axis variables
	
	SLT1_P1_050_DI01 	: FB_EL1809;
	SLT1_P1_050_DI02 	: FB_EL1809;
	SLT1_P1_050_DI03 	: FB_EL1809;
	SLT1_P1_050_DI04 	: FB_EL1809;
	SLT1_P1_050_DI05 	: FB_EL1809;
	SLT1_P1_050_DI06 	: FB_EL1809;

	SLT1_P1_050_DO01 	: FB_EL2809;
	SLT1_P1_050_DO02 	: FB_EL2809;
	SLT1_P1_050_DO03 	: FB_EL2809;
	SLT1_P1_050_DO04 	: FB_EL2809;
	SLT1_P1_050_DO05 	: FB_EL2809;
	SLT1_P1_050_DO06 	: FB_EL2809;	

	
	ARK_P1_050_DI01     : FB_EL1809;        // Digital inputs card
    ARK_P1_050_DO01     : FB_EL2809;        // Digital outputs card	
    ARK_P1_050_DO02     : FB_EL2809;        // Digital outputs card			
    ARK_P1_050_AI01     : FB_EL3002;        // Digital outputs card
    ARK_P1_050_AO01     : FB_EL4004;        // Digital outputs card		
    ARK_P1_050_AO02     : FB_EL4004;        // Digital outputs card		

	STK_P2_050_AO1	: FB_EL4004;	
	STK_P2_050_DI1	: FB_EL1809;	
	STK_P2_050_DI2	: FB_EL1809;	
	STK_P2_050_DO1	: FB_EL2809;	
	STK_P2_050_DO2	: FB_EL2809;	
	
	
	STK_P2_050_AO2	: FB_EL4004;	
	STK_P2_050_AO3	: FB_EL4004;	
	STK_P2_050_AO4	: FB_EL4004;	

	STK_P2_050_ENC1 : FB_EL5152;
	//Io-Link master
	STK_050_BC2	: _FB_006B51;
	//Io-Link Slaves
	STKL_050_DIO1 : _FB_00BE31;	//Ch 0 - IO-Link IP67 Input/Output module
	STKL_050_DIO2 : _FB_00BH11; //Ch 1 - IO-Link DIN Rail Input/Output module
	STKL_100_B01 : _FB_DT35_B15251; //Ch 2 - IO-Link Pile height sensor	
	
	STKU_050_DIO1 : _FB_00BH11; //Ch 1 - IO-Link DIN Rail Input/Output module
	STKU_050_DIO2 : _FB_00BH11; //Ch 1 - IO-Link DIN Rail Input/Output module
	STKU_050_DIO3 : _FB_00BH11; //Ch 1 - IO-Link DIN Rail Input/Output module
	
	STKU_P2_100_UG8 : FB_IS620P_CO; //Backstop servo drive
	STKU_P2_100_UG9 : FB_IS620P_CO; //Lift servo drive

	statusWord AT %I* : UINT;
	
    STK_P2_050_SP01     : FB_EL6910;        // Safety processor (TwinSAFE)	
	ARK_P1_050_DI02     : FB_EL1008;        // Digital inputs card	
END_VAR

// ---- GVLs/GVL_InterConnection.TcGVL
{attribute 'Tc2GvlVarNames'}
VAR_GLOBAL
	
	upperStackerUnload : BOOL;
	lowerStackerUnload : BOOL;
	upperStackerExternalCounterReset : BOOL;
	lowerStackerExternalCounterReset : BOOL;

END_VAR

// ---- POUs/FAST.TcPOU
PROGRAM FAST
VAR
	instFB_MetricsAndCalculation: FB_MetricsAndCalculation;
	
END_VAR

_00_UpdateHardware();
_03_MetricsAndCalculation();

(*==============================================================================================================================
CPNTeck - Automação industrial
(c)Copyright 2023 All Rights Reserved
_______________________________________________________________________________________________________________________________
Library: <N/A or library name>
Tested with: <PLC / IPC model>
Engineering: <TwinCAT version>
Restrictions: <text>
Requirements: <text>
Functionality: <short description>
Support: <email>
Note: Parameter comments are only available in language 'English (United States)'
_______________________________________________________________________________________________________________________________
Change log table:

Version  		| Date        			| Expert in charge  	| Changes applied
<xx.xx.xx>		| <dd.mm.yyyy>  		| <name>              | <changes>

===============================================================================================================================*)

METHOD _00_UpdateHardware
VAR_INPUT
END_VAR
SLT1_P1_050_DI01();
SLT1_P1_050_DI02();
SLT1_P1_050_DI03();
SLT1_P1_050_DI04();
SLT1_P1_050_DI05();
SLT1_P1_050_DI06();

SLT1_P1_050_DO01();
SLT1_P1_050_DO02();
SLT1_P1_050_DO03();
SLT1_P1_050_DO04();
SLT1_P1_050_DO05();
SLT1_P1_050_DO06();

ARK_P1_050_DI01();
ARK_P1_050_DI02();
ARK_P1_050_DO01();
ARK_P1_050_DO02();

ARK_P1_050_AI01();
ARK_P1_050_AO01();	
ARK_P1_050_AO02();
END_METHOD

METHOD _03_MetricsAndCalculation
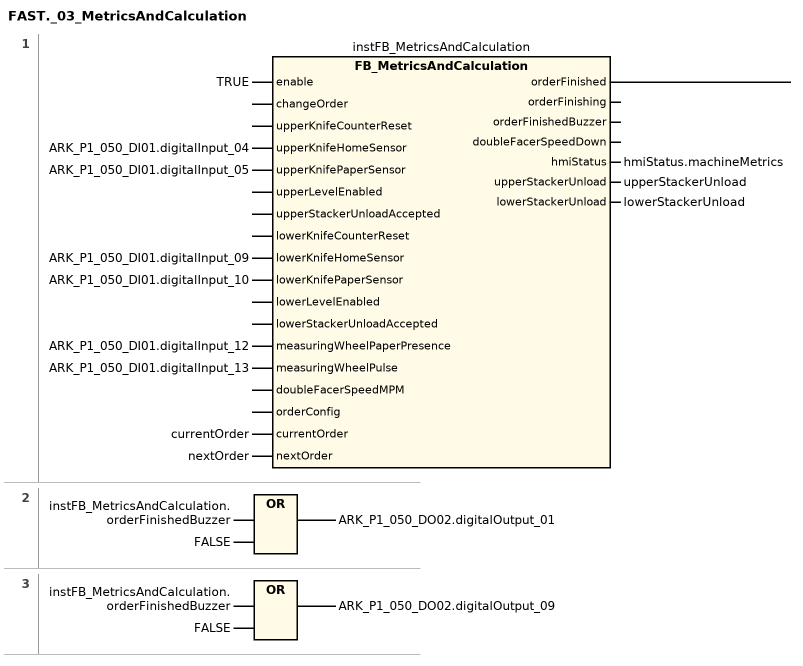
// NETWORK 1
instFB_MetricsAndCalculation(
    enable := TRUE,
    upperKnifeHomeSensor := ARK_P1_050_DI01.digitalInput_04,
    upperKnifePaperSensor := ARK_P1_050_DI01.digitalInput_05,
    lowerKnifeHomeSensor := ARK_P1_050_DI01.digitalInput_09,
    lowerKnifePaperSensor := ARK_P1_050_DI01.digitalInput_10,
    measuringWheelPaperPresence := ARK_P1_050_DI01.digitalInput_12,
    measuringWheelPulse := ARK_P1_050_DI01.digitalInput_13,
    currentOrder := currentOrder,
    nextOrder := nextOrder,
    hmiStatus => hmiStatus.machineMetrics,
    upperStackerUnload => upperStackerUnload,
    lowerStackerUnload => lowerStackerUnload); // FB_MetricsAndCalculation

// NETWORK 2
ARK_P1_050_DO02.digitalOutput_01 := instFB_MetricsAndCalculation.orderFinishedBuzzer OR FALSE;

// NETWORK 3
ARK_P1_050_DO02.digitalOutput_09 := instFB_MetricsAndCalculation.orderFinishedBuzzer OR FALSE;
END_METHOD

END_PROGRAM

// ---- Library/Machine/DryEnd/Order control/FB_MetricsAndCalculation.TcPOU
FUNCTION_BLOCK FB_MetricsAndCalculation

//======================================================================
// INPUTS
//======================================================================
VAR_INPUT

    //────────────────────────────────────────────
    // GENERAL CONTROL
    //────────────────────────────────────────────
    enable                          : BOOL;   // FB enable
    changeOrder                     : BOOL;   // Request order change

    //────────────────────────────────────────────
    // UPPER KNIFE / LEVEL — COUNTERS & SENSORS
    //────────────────────────────────────────────
    upperKnifeCounterReset          : BOOL;   // Upper level sheet counter reset
    upperKnifeHomeSensor            : BOOL;   // Upper level home sensor (counter pulse)
    upperKnifePaperSensor   		: BOOL;   // Upper level paper presence
    upperLevelEnabled               : BOOL;   // Upper level enabled

    // EN: External upper-level command that resets only the active pile quantity.
    // PT: Comando externo do nível superior que zera somente a quantidade da pilha ativa.
    upperStackerUnloadAccepted      : BOOL;

    //────────────────────────────────────────────
    // LOWER KNIFE / LEVEL — COUNTERS & SENSORS
    //────────────────────────────────────────────
    lowerKnifeCounterReset          : BOOL;   // Lower level sheet counter reset
    lowerKnifeHomeSensor            : BOOL;   // Lower level home sensor (counter pulse)
    lowerKnifePaperSensor   		: BOOL;   // Lower level paper presence
    lowerLevelEnabled               : BOOL;   // Lower level enabled

    // EN: External lower-level command that resets only the active pile quantity.
    // PT: Comando externo do nível inferior que zera somente a quantidade da pilha ativa.
    lowerStackerUnloadAccepted      : BOOL;

    //────────────────────────────────────────────
    // MEASURING WHEEL
    //────────────────────────────────────────────
    measuringWheelPaperPresence     : BOOL;   // Paper presence at measuring wheel
    measuringWheelPulse        : BOOL;   // Measuring wheel pulse counter

    //────────────────────────────────────────────
    // MACHINE SPEED / CONFIGURATION
    //────────────────────────────────────────────
    doubleFacerSpeedMPM             : REAL;   // Double facer speed [m/min]
    orderConfig                     : orderConfig_TypeStruct;

END_VAR


//======================================================================
// OUTPUTS
//======================================================================
VAR_OUTPUT

    //────────────────────────────────────────────
    // ORDER STATUS
    //────────────────────────────────────────────
    orderFinished                   : BOOL;   // Order completed
    orderFinishing                  : BOOL;   // Order in finishing phase
	orderFinishedBuzzer				: BOOL;
	
    //────────────────────────────────────────────
    // MACHINE CONTROL
    //────────────────────────────────────────────
    doubleFacerSpeedDown            : BOOL;   // Request speed reduction

    //────────────────────────────────────────────
    // HMI
    //────────────────────────────────────────────
    hmiStatus                       : orderHmiStatus_TypeStruct;
	
    //────────────────────────────────────────────
    // EXT COMMANDS
    //────────────────────────────────────────────

    // EN: Timed automatic unload pulse for the upper stacker.
    // PT: Pulso temporizado de descarte automático do stacker superior.
	upperStackerUnload		: BOOL;

    // EN: Timed automatic unload pulse for the lower stacker.
    // PT: Pulso temporizado de descarte automático do stacker inferior.
	lowerStackerUnload		: BOOL;

END_VAR


//======================================================================
// INTERNAL VARIABLES
//======================================================================
VAR

    // EN: Extends automatic unload requests for external stacker interfaces.
    // PT: Prolonga os pedidos automáticos para interfaces de stackers externos.
    instTPUpperStackerUnload        : TP;
    instTPLowerStackerUnload        : TP;

    //────────────────────────────────────────────
    // EDGE DETECTION / STATE
    //────────────────────────────────────────────
    changeOrderOld                  : BOOL;

    upperLevelHomeSensorOld         : BOOL;
    lowerLevelHomeSensorOld         : BOOL;

    // EN: External pile reset commands are processed only on rising edges.
    // PT: Os comandos externos de reset da pilha são processados somente nas bordas de subida.
    upperStackerResetOld            : BOOL;
    lowerStackerResetOld            : BOOL;
    rUpperStackerReset              : BOOL;
    rLowerStackerReset              : BOOL;

    //────────────────────────────────────────────
    // SHEET COUNTERS
    //────────────────────────────────────────────
    upperKnifelSheetCounter          : DINT;
    lowerKnifeSheetCounter          : DINT;

    //────────────────────────────────────────────
    // MEASURING WHEEL
    //────────────────────────────────────────────
    measuringWheelPulseOld     : BOOL;

    //────────────────────────────────────────────
    // TIME / SYSTEM
    //────────────────────────────────────────────
    instFBLocalSystemTime           : FB_LocalSystemTime;
    instFBGetTimeZoneInformation    : FB_GetTimeZoneInformation;
    localTimeZone                   : Tc2_Utilities.E_TimeZoneID;

    instClkProg1Min                 : CLK_PRG;    // 1-minute clock pulse

    //────────────────────────────────────────────
    // INDEXES / STATE MACHINES
    //────────────────────────────────────────────
    index                           : INT;
    resetIndex                     : INT;
    count                           : INT;

    notRunningTimeIndex             : INT;
    linearMetersCalculationIndex    : INT;
    averageSpeedIndex               : INT;

    //────────────────────────────────────────────
    // SPEED STATISTICS (RUNTIME)
    //────────────────────────────────────────────
    arrAverageSpeedPerHour          : ARRAY [0..23] OF INT; // Avg speed per hour

	instTON_SaveSQLTimeOut: TON;
	instGEN_PULSEBuzzer: GEN_PULSE;
	changeOrderRequestOld: BOOL;
	instGEN_PULSEPlcWatchDog: GEN_PULSE;	
	
END_VAR


//======================================================================
// PERSISTENT DATA
//======================================================================
VAR PERSISTENT

    //────────────────────────────────────────────
    // PRODUCTION METRICS (PER HOUR)
    //────────────────────────────────────────────
    arrMetersPerHour                : ARRAY [0..23] OF INT; // Produced meters per hour
    arrPulsePerHour                 : ARRAY [0..23] OF INT; // Measuring wheel pulses per hour
    arrMachineNotRunningTimePerHour : ARRAY [0..23] OF INT; // Machine stopped time per hour

    wDayOfWeekOld                   : WORD; // Used to detect day change

END_VAR


//======================================================================
// IN/OUT VARIABLES
//======================================================================
VAR_IN_OUT

    currentOrder                    : Order_TypeStruct;
    nextOrder                       : Order_TypeStruct;

END_VAR

(*=================================================================================================
CPNTeck - Automação ind.
(c)Copyright 2022 All Rights Reserved
_______________________________________________________________________________________________________________________________
Library: N/A 
Tested with: CX5140 
Engineering: Twincat 2
Restrictions: -
Requirements: N/A
Functionality: This function block offers basic functionalities to control the order and count the varibles
the fallowing functions:
- Reduce the double facer speed
- Execute a single cut in the material web
- Increase the speed of the dryend
- Change the slitter order
- Change the rotary knife sheet lenght
- Execute the stacker discharge of the remaining boards
- Increase the speed of the double facer the the speed that it was before.

Support: fabio@cpnteck.com.br
Note: Parameter comments are only available in language 'English (United States)'
_______________________________________________________________________________________________________________________________
Change log table:
Version  		| Date        			| Expert in charge  			| Changes applied

01.00.01		| 28.09.2022  		| Fabio Campion                	| First released version



==================================================================================================*)

ACT_OneMinuteClock();
ACT_AverageSpeedPerHourCalculation();
ACT_ProgramCurrentOrder();
ACT_SheetCounter();
ACT_OderStatusDisplay();
ACT_MetersPerHourCalculation();
ACT_MachineNotRunningTimePerHour();
ACT_ResetMetrics();
_01_LinearMetersCalculation();
_012_ChangeOrder();
_13_PlcWatchDog();

instFBGetTimeZoneInformation(bExecute := TRUE);
instFBLocalSystemTime(bEnable := TRUE, dwCycle := 1);

METHOD _01_LinearMetersCalculation
VAR
    kMmToM : REAL := 0.001; // mm → m conversion factor
    // Working variables
    rProd1 : REAL;
    rTot1  : REAL;
    rRem1  : REAL;

    rProd2 : REAL;
    rTot2  : REAL;
    rRem2  : REAL;
END_VAR
//==============================================================
// CUTS REMAINING (PER ORDER) — ALWAYS UPDATED WHEN RELEVANT
//==============================================================
currentOrder.order1.numberOfCutsRemaining := currentOrder.order1.numberOfCuts - currentOrder.order1.numberOfCutsProduced;
currentOrder.order2.numberOfCutsRemaining := currentOrder.order2.numberOfCuts - currentOrder.order2.numberOfCutsProduced;		


//==============================================================
// LINEAR METERS CALCULATION
// Formula (per order):
//   total     = sheetLength[mm] * 0.001 * numberOfCuts
//   produced  = sheetLength[mm] * 0.001 * numberOfCutsProduced
//   remaining = total - produced
//==============================================================
CASE currentOrder.levelSelector OF

    //==========================================================
    // ORDER 1 ONLY (Upper level -> Order 1)
    //==========================================================
    E_LevelSelector.eUpperOnly:

        rProd1 := (currentOrder.order1.sheetLength * kMmToM) * currentOrder.order1.numberOfCutsProduced;
        rTot1  := (currentOrder.order1.sheetLength * kMmToM) * currentOrder.order1.numberOfCuts;
        rRem1  := rTot1 - rProd1;

        currentOrder.linearMetersProduced  := rProd1;
        currentOrder.linearMetersRemaining := rRem1;
        currentOrder.linearMeters          := rTot1;


    //==========================================================
    // ORDER 1 ONLY (Lower level -> Order 1)  // corrected mapping
    //==========================================================
    E_LevelSelector.eLowerOnly:

        rProd1 := (currentOrder.order1.sheetLength * kMmToM) * currentOrder.order1.numberOfCutsProduced;
        rTot1  := (currentOrder.order1.sheetLength * kMmToM) * currentOrder.order1.numberOfCuts;
        rRem1  := rTot1 - rProd1;

        currentOrder.linearMetersProduced  := rProd1;
        currentOrder.linearMetersRemaining := rRem1;
        currentOrder.linearMeters          := rTot1;


    //==========================================================
    // BOTH ORDERS (SUM)
    // Order 1 uses LOWER counter (but order1 parameters)
    // Order 2 uses UPPER counter (but order2 parameters)
    //==========================================================
    E_LevelSelector.eBoth:

        // Order 1 (Lower level -> Order 1)
        rProd1 := (currentOrder.order1.sheetLength * kMmToM) * currentOrder.order1.numberOfCutsProduced;
        rTot1  := (currentOrder.order1.sheetLength * kMmToM) * currentOrder.order1.numberOfCuts;
        rRem1  := rTot1 - rProd1;

        // Order 2 (Upper level -> Order 2)
        rProd2 := (currentOrder.order2.sheetLength * kMmToM) * currentOrder.order2.numberOfCutsProduced;
        rTot2  := (currentOrder.order2.sheetLength * kMmToM) * currentOrder.order2.numberOfCuts;
        rRem2  := rTot2 - rProd2;

        // Aggregate totals for overall order
        currentOrder.linearMetersProduced  := rProd1;
        currentOrder.linearMetersRemaining := rRem1;
        currentOrder.linearMeters          := rTot1;

		

		
END_CASE
END_METHOD

METHOD _012_ChangeOrder
VAR_INPUT
END_VAR

VAR

	
END_VAR

//Reset the saved flag 
IF currentOrder.changeOrderRequest AND NOT changeOrderRequestOld THEN
	
	currentOrder.saveSQLFinished := FALSE;

END_IF

changeOrderRequestOld := currentOrder.changeOrderRequest;


IF (currentOrder.changeOrderRequest AND currentOrder.saveSQLFinished) OR  currentOrder.saveSQLTimeOut THEN
	
	currentOrder.startedAt           	:= nextOrder.startedAt;
	currentOrder.tableID             	:= nextOrder.tableID;
	currentOrder.productionListNumber 	:= nextOrder.productionListNumber;
	currentOrder.paperComposition  	  	:= nextOrder.paperComposition;
	currentOrder.fluteType           	:= nextOrder.fluteType;
	currentOrder.paperWidth          	:= nextOrder.paperWidth;
	currentOrder.paper1              	:= nextOrder.paper1;
	currentOrder.paper2              	:= nextOrder.paper2;
	currentOrder.paper3              	:= nextOrder.paper3;
	currentOrder.paper4              	:= nextOrder.paper4;
	currentOrder.paper5              	:= nextOrder.paper5;
	currentOrder.linearMeters        	:= nextOrder.linearMeters;
	currentOrder.linearMetersProduced 	:= nextOrder.linearMetersProduced;
	currentOrder.linearMetersRemaining	:= nextOrder.linearMeters;
	currentOrder.scorerHeightMM      	:= nextOrder.scorerHeightMM;
	currentOrder.levelSelector       	:= nextOrder.levelSelector;
	currentOrder.invertOrderLevel    	:= nextOrder.invertOrderLevel;
	currentOrder.invertOrderSide     	:= nextOrder.invertOrderSide;
	currentOrder.order1              	:= nextOrder.order1;
	currentOrder.order2              	:= nextOrder.order2;
	currentOrder.aocRequest             := nextOrder.aocRequest;
	currentOrder.changeOrderRequest     := nextOrder.changeOrderRequest;

END_IF

instTON_SaveSQLTimeOut(IN := currentOrder.changeOrderRequest, PT:= T#5S, Q=>currentOrder.saveSQLTimeOut );
END_METHOD

METHOD _13_PlcWatchDog
VAR_INPUT
END_VAR

VAR

END_VAR

instGEN_PULSEPlcWatchDog(
    ENQ := TRUE,
    PTH := T#500MS,
    PTL := T#500MS
);

currentOrder.plcWatchDog := instGEN_PULSEPlcWatchDog.Q;
END_METHOD

ACTION ACT_AverageSpeedPerHourCalculation:
//----------------------------------------------------------------------------------------------
// Calculate the machine average speed per hour
// Converts meters per hour into meters per minute for each hour slot (0 to 23)
//----------------------------------------------------------------------------------------------
FOR averageSpeedIndex := 0 TO 23 BY 1 DO
	
	IF arrMetersPerHour[averageSpeedIndex] > 0 THEN
		arrAverageSpeedPerHour[averageSpeedIndex] := arrMetersPerHour[averageSpeedIndex] / 60;
	ELSE
		arrAverageSpeedPerHour[averageSpeedIndex] := 0;
	END_IF

END_FOR

//----------------------------------------------------------------------------------------------
// Update HMI status structure with calculated average speeds
//----------------------------------------------------------------------------------------------
hmiStatus.arrAverageSpeedPerHour := arrAverageSpeedPerHour;
END_ACTION

ACTION ACT_MachineNotRunningTimePerHour:
//----------------------------------------------------------------------------------------------
// Calculate stop time per hour and total machine stopped time for the order
// If the machine speed is below 20 MPM, count it as downtime
//----------------------------------------------------------------------------------------------
IF instClkProg1Min.Q AND doubleFacerSpeedMPM < 20 THEN
	
	// Increment downtime for the current hour
	arrMachineNotRunningTimePerHour[index] := arrMachineNotRunningTimePerHour[index] + 1;

	// Reset total downtime accumulator before recalculating
	hmiStatus.machineNotRunningTimeTotal := 0;

	//------------------------------------------------------------------------------------------
	// Sum all hourly downtime values to get total machine stopped time
	//------------------------------------------------------------------------------------------
	FOR notRunningTimeIndex := 0 TO 23 BY 1 DO
		hmiStatus.machineNotRunningTimeTotal := hmiStatus.machineNotRunningTimeTotal + arrMachineNotRunningTimePerHour[notRunningTimeIndex];
	END_FOR

END_IF

//----------------------------------------------------------------------------------------------
// Update HMI structure with current hourly machine stop time array
//----------------------------------------------------------------------------------------------
hmiStatus.arrMachineNotRunningTimePerHour := arrMachineNotRunningTimePerHour;
END_ACTION

ACTION ACT_MetersPerHourCalculation:
//----------------------------------------------------------------------------------------------
// Calculate the linear meters produced per hour
// Uses measuring wheel pulses and wheel diameter to compute distance
//----------------------------------------------------------------------------------------------

// Get the current hour index from system time
index := WORD_TO_INT(instFBLocalSystemTime.systemTime.wHour);

//----------------------------------------------------------------------------------------------
// Detect pulse from measuring wheel when paper is present
//----------------------------------------------------------------------------------------------
IF measuringWheelPulse AND NOT measuringWheelPulseOld AND measuringWheelPaperPresence THEN

	// Increment pulse count for the current hour
	arrPulsePerHour[index] := arrPulsePerHour[index] + 1;

	// Convert pulse count to meters using wheel diameter
	arrMetersPerHour[index] := REAL_TO_INT(arrPulsePerHour[index] * ((orderConfig.measuringWheelDiameter * 3.14) * 0.001));

	// Reset linear meters accumulator before summing
	hmiStatus.linearMetersProduced := 0;

	//------------------------------------------------------------------------------------------
	// Sum linear meters produced for all hours to get total production
	//------------------------------------------------------------------------------------------
	FOR linearMetersCalculationIndex := 0 TO 23 BY 1 DO
		hmiStatus.linearMetersProduced := hmiStatus.linearMetersProduced + arrMetersPerHour[linearMetersCalculationIndex];
	END_FOR

END_IF

//----------------------------------------------------------------------------------------------
// Store current pulse counter for next edge detection cycle
//----------------------------------------------------------------------------------------------
measuringWheelPulseOld := measuringWheelPulse;

//----------------------------------------------------------------------------------------------
// Update HMI with meters produced per hour
//----------------------------------------------------------------------------------------------
hmiStatus.arrMetersPerHour := arrMetersPerHour;
END_ACTION

ACTION ACT_OderStatusDisplay:
//----------------------------------------------------------------------------------------------
// Display an alert when the order is almost finishing
// Triggered when remaining linear meters are below a configured threshold
//----------------------------------------------------------------------------------------------
IF currentOrder.linearMetersRemaining < orderConfig.orderFinishingAlertWhenRemainig THEN
	orderFinishing := TRUE;
	hmiStatus.orderFinishing := TRUE;
ELSE
	orderFinishing := FALSE;
	hmiStatus.orderFinishing := FALSE;
END_IF

//----------------------------------------------------------------------------------------------
// Display an alert when the order is finished
// Triggered when there are no remaining linear meters to produce
//----------------------------------------------------------------------------------------------
IF currentOrder.linearMetersRemaining <= 0 THEN
	orderFinished := TRUE;
	hmiStatus.orderFinished := TRUE;
ELSE
	orderFinished := FALSE;
	hmiStatus.orderFinished := FALSE;
END_IF

// Pulse generator for DF speed up/down buttons
instGEN_PULSEBuzzer(
    ENQ := TRUE,
    PTH := T#1M,
    PTL := T#2M
);

orderFinishedBuzzer := orderFinishing AND instGEN_PULSEBuzzer.Q;
END_ACTION

ACTION ACT_OneMinuteClock:
//----------------------------------------------------------------------------------------------
// One-minute clock
// Used to calculate machine not running time and time-based counters
//----------------------------------------------------------------------------------------------
instClkProg1Min(PT := T#1M);

//----------------------------------------------------------------------------------------------
// Increment counter every time the one-minute timer elapses
//----------------------------------------------------------------------------------------------
IF instClkProg1Min.Q THEN
	count := count + 1;
END_IF
END_ACTION

ACTION ACT_ProgramCurrentOrder:
//----------------------------------------------------------------------------------------------
// Load next order when changeOrder is triggered (rising edge)
//----------------------------------------------------------------------------------------------
IF changeOrder AND NOT changeOrderOld THEN
	currentOrder := nextOrder;
END_IF

//----------------------------------------------------------------------------------------------
// Store previous state of changeOrder for edge detection
//----------------------------------------------------------------------------------------------
changeOrderOld := changeOrder;
END_ACTION

ACTION ACT_ResetMetrics:
//----------------------------------------------------------------------------------------------
// Reset metric arrays once per day (on day change)
//----------------------------------------------------------------------------------------------
IF instFBLocalSystemTime.systemTime.wDayOfWeek <> wDayOfWeekOld THEN

	//------------------------------------------------------------------------------------------
	// Clear all hourly tracking arrays (pulses, meters, downtime, average speed)
	//------------------------------------------------------------------------------------------
	FOR resetIndex := 0 TO 23 BY 1 DO
		arrPulsePerHour[resetIndex] := 0;
		arrMetersPerHour[resetIndex] := 0;
		arrMachineNotRunningTimePerHour[resetIndex] := 0;
		arrAverageSpeedPerHour[resetIndex] := 0;
	END_FOR

	//------------------------------------------------------------------------------------------
	// Store the current day to detect next change
	//------------------------------------------------------------------------------------------
	wDayOfWeekOld := instFBLocalSystemTime.systemTime.wDayOfWeek;

END_IF
END_ACTION

ACTION ACT_SheetCounter:
//==========================================================
// 1) Default automatic unload triggers
//==========================================================
// EN: These one-scan triggers are extended by the TP instances at the end.
// PT: Estes gatilhos de um scan são prolongados pelas instâncias TP ao final.
upperStackerUnload := FALSE;
lowerStackerUnload := FALSE;


//==========================================================
// 2) External pile reset edge detection
//==========================================================
// EN: Process each external reset only once, even if it remains TRUE for
//     several FAST-task scans.
// PT: Processa cada reset externo somente uma vez, mesmo que permaneça TRUE
//     durante vários scans da tarefa FAST.
rUpperStackerReset :=
    upperStackerUnloadAccepted AND NOT upperStackerResetOld;

rLowerStackerReset :=
    lowerStackerUnloadAccepted AND NOT lowerStackerResetOld;

upperStackerResetOld := upperStackerUnloadAccepted;
lowerStackerResetOld := lowerStackerUnloadAccepted;


//==========================================================
// 3) Reset only the pile quantity selected for each level
//==========================================================
// EN: Reset is performed before sheet counting. A valid sheet edge in the
//     same scan therefore becomes the first sheet of the new pile.
// PT: O reset é executado antes da contagem. Uma borda válida de chapa no
//     mesmo scan passa a ser a primeira chapa da nova pilha.
CASE currentOrder.levelSelector OF

    E_LevelSelector.eUpperOnly:
        IF rUpperStackerReset THEN
            currentOrder.order1.pileQuantityProduced := 0;
        END_IF

    E_LevelSelector.eLowerOnly:
        IF rLowerStackerReset THEN
            currentOrder.order1.pileQuantityProduced := 0;
        END_IF

    E_LevelSelector.eBoth:
        IF rLowerStackerReset THEN
            currentOrder.order1.pileQuantityProduced := 0;
        END_IF

        IF rUpperStackerReset THEN
            currentOrder.order2.pileQuantityProduced := 0;
        END_IF

END_CASE;


//==========================================================
// 4) Sheet counting
//==========================================================
CASE currentOrder.levelSelector OF

    //==========================================================
    // ORDER 1 ONLY
    // Upper level -> Order 1
    //==========================================================
    E_LevelSelector.eUpperOnly:

        // EN: Count one valid upper knife home-sensor rising edge.
        // PT: Conta uma borda de subida válida do sensor de home da faca superior.
        IF upperKnifeHomeSensor AND NOT upperLevelHomeSensorOld AND upperKnifePaperSensor THEN

            upperKnifelSheetCounter := upperKnifelSheetCounter + 1;
            currentOrder.order1.numberOfCutsProduced :=
                currentOrder.order1.numberOfCutsProduced + 1;
            currentOrder.order1.pileQuantityProduced :=
                currentOrder.order1.pileQuantityProduced + 1;

        END_IF

        upperLevelHomeSensorOld := upperKnifeHomeSensor;


    //==========================================================
    // ORDER 1 ONLY
    // Lower level -> Order 1
    //==========================================================
    E_LevelSelector.eLowerOnly:

        // EN: Count one valid lower knife home-sensor rising edge.
        // PT: Conta uma borda de subida válida do sensor de home da faca inferior.
        IF lowerKnifeHomeSensor AND NOT lowerLevelHomeSensorOld AND lowerKnifePaperSensor THEN

            currentOrder.order1.numberOfCutsProduced :=
                currentOrder.order1.numberOfCutsProduced + 1;
            currentOrder.order1.pileQuantityProduced :=
                currentOrder.order1.pileQuantityProduced + 1;

        END_IF

        lowerLevelHomeSensorOld := lowerKnifeHomeSensor;


    //==========================================================
    // BOTH ORDERS
    // Order 1 uses lower level
    // Order 2 uses upper level
    //==========================================================
    E_LevelSelector.eBoth:

        //======================================================
        // ORDER 1
        // Lower level -> Order 1
        //======================================================
        IF lowerKnifeHomeSensor AND NOT lowerLevelHomeSensorOld AND lowerKnifePaperSensor THEN

            currentOrder.order1.numberOfCutsProduced :=
                currentOrder.order1.numberOfCutsProduced + 1;
            currentOrder.order1.pileQuantityProduced :=
                currentOrder.order1.pileQuantityProduced + 1;

        END_IF


        //======================================================
        // ORDER 2
        // Upper level -> Order 2
        //======================================================
        IF upperKnifeHomeSensor AND NOT upperLevelHomeSensorOld AND upperKnifePaperSensor THEN

            upperKnifelSheetCounter := upperKnifelSheetCounter + 1;
            currentOrder.order2.numberOfCutsProduced :=
                currentOrder.order2.numberOfCutsProduced + 1;
            currentOrder.order2.pileQuantityProduced :=
                currentOrder.order2.pileQuantityProduced + 1;

        END_IF

        lowerLevelHomeSensorOld := lowerKnifeHomeSensor;
        upperLevelHomeSensorOld := upperKnifeHomeSensor;

END_CASE;


//==========================================================
// 5) Order 1 full counter reset
//==========================================================
// EN: Existing order reset keeps its original full-reset behavior.
// PT: O reset existente da ordem mantém seu comportamento de reset completo.
IF currentOrder.order1.counterReset THEN
    currentOrder.order1.numberOfCutsProduced := 0;
    currentOrder.order1.pileQuantityProduced := 0;
    currentOrder.order1.pileCounter := 0;
    currentOrder.order1.pileQuantityRemaining := 0;

END_IF;


//==========================================================
// 6) Order 2 full counter reset
//==========================================================
// EN: Existing order reset keeps its original full-reset behavior.
// PT: O reset existente da ordem mantém seu comportamento de reset completo.
IF currentOrder.order2.counterReset THEN
    currentOrder.order2.numberOfCutsProduced := 0;
    currentOrder.order2.pileQuantityProduced := 0;
    currentOrder.order2.pileCounter := 0;
    currentOrder.order2.pileQuantityRemaining := 0;

END_IF;


//==========================================================
// 7) Close completed piles and trigger automatic unload
//==========================================================
// EN: Reaching the configured quantity closes and resets the pile immediately;
//     it also generates the unload trigger for the selected level.
// PT: Atingir a quantidade configurada fecha e zera a pilha imediatamente;
//     também gera o gatilho de descarte para o nível selecionado.
CASE currentOrder.levelSelector OF

    E_LevelSelector.eUpperOnly:
        IF (currentOrder.order1.pileQuantity > 0) AND
           (currentOrder.order1.pileQuantityProduced >= currentOrder.order1.pileQuantity) THEN

            currentOrder.order1.pileQuantityProduced := 0;
            currentOrder.order1.pileCounter :=
                currentOrder.order1.pileCounter + 1;
            upperStackerUnload := TRUE;

            IF currentOrder.order1.pileQuantityRemaining > 0 THEN
                currentOrder.order1.pileQuantityRemaining :=
                    currentOrder.order1.pileQuantityRemaining - 1;
            END_IF

        END_IF

    E_LevelSelector.eLowerOnly:
        IF (currentOrder.order1.pileQuantity > 0) AND
           (currentOrder.order1.pileQuantityProduced >= currentOrder.order1.pileQuantity) THEN

            currentOrder.order1.pileQuantityProduced := 0;
            currentOrder.order1.pileCounter :=
                currentOrder.order1.pileCounter + 1;
            lowerStackerUnload := TRUE;

            IF currentOrder.order1.pileQuantityRemaining > 0 THEN
                currentOrder.order1.pileQuantityRemaining :=
                    currentOrder.order1.pileQuantityRemaining - 1;
            END_IF

        END_IF

    E_LevelSelector.eBoth:
        IF (currentOrder.order1.pileQuantity > 0) AND
           (currentOrder.order1.pileQuantityProduced >= currentOrder.order1.pileQuantity) THEN

            currentOrder.order1.pileQuantityProduced := 0;
            currentOrder.order1.pileCounter :=
                currentOrder.order1.pileCounter + 1;
            lowerStackerUnload := TRUE;

            IF currentOrder.order1.pileQuantityRemaining > 0 THEN
                currentOrder.order1.pileQuantityRemaining :=
                    currentOrder.order1.pileQuantityRemaining - 1;
            END_IF

        END_IF

        IF (currentOrder.order2.pileQuantity > 0) AND
           (currentOrder.order2.pileQuantityProduced >= currentOrder.order2.pileQuantity) THEN

            currentOrder.order2.pileQuantityProduced := 0;
            currentOrder.order2.pileCounter :=
                currentOrder.order2.pileCounter + 1;
            upperStackerUnload := TRUE;

            IF currentOrder.order2.pileQuantityRemaining > 0 THEN
                currentOrder.order2.pileQuantityRemaining :=
                    currentOrder.order2.pileQuantityRemaining - 1;
            END_IF

        END_IF

END_CASE;


